FUNCTION_BLOCK FB_BA_WeatherStation EXTENDS FB_BA_View
VAR_INPUT
END_VAR
VAR_OUTPUT
END_VAR
VAR
	WeatherStation				: FB_BA_RawPublisher;
	stWeatherStation			: ST_BA_WeatherStation;
END_VAR

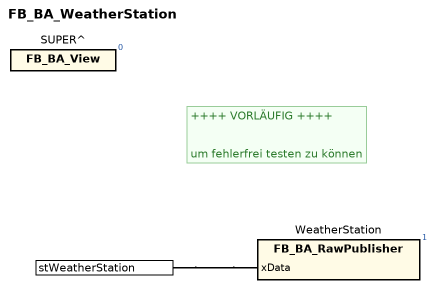
SUPER^(); // FB_BA_View
// ++++ VORLÄUFIG ++++
//
// um fehlerfrei testen zu können
WeatherStation(xData := stWeatherStation); // FB_BA_RawPublisher

END_FUNCTION_BLOCK

(* stored: Version 1.1.0.1, ProductVersion 3.1.4024.6
   POU FB_BA_WeatherStation: Id {74f6ee1c-6733-46e8-9b4e-802319917a80}, SpecialFunc None *)
